(* PLC project CoDeSys External Library Template, WAGO e!COCKPIT e!COCKPIT, author 3S - Smart Software Solutions GmbH *)
(* stored: creationDateTime 2019-10-29T12:22:40.3456623, version 3.5.5.30, modificationDateTime 2019-10-24T14:40:07.960949, organization 3S - Smart Software Solutions GmbH *)
(* Library project template with all possible element types, docu and a sample project structure *)

(* values of enumPPPSBramkaSTC65RS485ModbusError: BrakKomunikacji: brak komunikacji (MODBUS RTU) z konwerterem; ResetKonwertera: reset konwertera; BrakTelegramowEnOcean: brak odbioru telegramów EnOcean (brak komunikacji EnOcean) *)

(* Autor: Paweł Kąkol, 2018-08-13-PK Prawa majątkowe: Solwena Sp. z o.o., Aktualizacje: 2018-09-10-PK - dodanie alarmów ResetKonwertera i BrakTelegramowEnOcean Opis: enum służy do obsługi alarmów w fb konwertera GTW0 na budynkach PPP Sopot *)
{attribute 'qualified_only'}
{attribute 'strict'}
TYPE enumPPPSBramkaSTC65RS485ModbusError : (BrakKomunikacji := 1, ResetKonwertera := 2, BrakTelegramowEnOcean := 3);
END_TYPE
